FUNCTION PENDING : BOOL
VAR_INPUT
	hr 	: DINT;
END_VAR
VAR
END_VAR

PENDING := hr = S_PENDING;

END_FUNCTION

(* stored: Version 1.1.0.1, ProductVersion 3.1.4026.18
   POU PENDING: Id {f539ec3a-bf13-4734-98a5-7ce796e4036d}, SpecialFunc None *)
